SEGMENT_TYPE EPL (* EPL Segment *)
  (* Standard: 61499 ITA; Description: Ethernet POWERLINK segment *)
  (* Version 0.1, 2012-06-18, 4DIAC-IDE, 4DIAC-Consortium *)
  VAR_INPUT
    Param : WSTRING; (* Param *)
  END_VAR
END_SEGMENT_TYPE
